# EPICS substitutions: iocBoot/iocvirPV/DPU05.substitutions
file "../../db/virAi.template"{ pattern
{DPU,	  num}
{05,	  0 }
{05,	  1 }
{05,	  2 }
{05,	  3 }
{05,	  4 }
{05,	  5 }
{05,	  6 }
{05,	  7 }
{05,	  8 }
{05,	  9 }
{05,	  10}
{05,	  11}
{05,	  12}
{05,	  13}
{05,	  14}
{05,	  15}
{05,	  16}
{05,	  17}
{05,	  18}
{05,	  19}
{05,	  20}
{05,	  21}
{05,	  22}
{05,	  23}
{05,	  24}
{05, 	  25}
{05,	  26}
{05,	  27}
{05,	  28}
{05,	  29}
{05,	  30}
{05,	  31}
{05,	  32}
{05,	  33}
{05,	  34}
{05,	  35}
{05,	  36}
{05,	  37}
{05,	  38}
{05,	  39}
{05,	  40}
{05,	  41}
{05,	  42}
{05,	  43}
{05,	  44}
{05,	  45}
{05,	  46}
{05,	  47}
{05,	  48}
{05,	  49}
{05,	  50}
{05,	  51}
{05,	  52}
{05,	  53}
{05,	  54}
{05,	  55}
{05,	  56}
{05,	  57}
{05,	  58}
{05,	  59}
{05,	  60}
{05,	  61}
{05,	  62}
{05, 	  63}
{05,      64}
{05,      65}
{05,      66}
{05,      67}
{05,      68}
{05,      69}
{05,      70}
{05,      71}
{05,      72}
{05,      73}
{05,      74}
{05,      75}
{05,      76}
{05,      77}
{05,      78}
{05,      79}
{05,      80}
{05,      81}
{05,      82}
{05,      83}
{05,      84}
{05,      85}
{05,      86}
{05,      87}
{05,      88}
{05,      89}
{05,      90}
{05,      91}
{05,      92}
{05,      93}
{05,      94}
{05,      95}
{05,      96}
{05,      97}
{05,      98}
{05,      99}
{05,     100}
{05,     101}
{05,     102}
{05,     103}
{05,     104}
{05,     105}
{05,     106}
{05,     107}
{05,     108}
{05,     109}
{05,     110}
{05,     111}
{05,     112}
{05,     113}
{05,     114}
{05,     115}
{05,     116}
{05,     117}
{05,     118}
{05,     119}
{05,     120}
{05,     121}
{05,     122}
{05,     123}
{05,     124}
{05,     125}
{05,     126}
{05,     127}
{05,     128}
{05,     129}
{05,     130}
{05,     131}
{05,     132}
{05,     133}
{05,     134}
{05,     135}
{05,     136}
{05,     137}
{05,     138}
{05,     139}
{05,     140}
{05,     141}
{05,     142}
{05,     143}
{05,     144}
{05,     145}
{05,     146}
{05,     147}
{05,     148}
{05,     149}
{05,     150}
{05,     151}
{05,     152}
{05,     153}
{05,     154}
{05,     155}
{05,     156}
{05,     157}
{05,     158}
{05,     159}
{05,     160}
{05,     161}
{05,     162}
{05,     163}
{05,     164}
{05,     165}
{05,     166}
{05,     167}
{05,     168}
{05,     169}
{05,     170}
{05,     171}
{05,     172}
{05,     173}
{05,     174}
{05,     175}
{05,     176}
{05,     177}
{05,     178}
{05,     179}
{05,     180}
{05,     181}
{05,     182}
{05,     183}
{05,     184}
{05,     185}
{05,     186}
{05,     187}
{05,     188}
{05,     189}
{05,     190}
{05,     191}
{05,     192}
{05,     193}
{05,     194}
{05,     195}
{05,     196}
{05,     197}
{05,     198}
{05,     199}
}
